FUNCTION_BLOCK FB_Cinta_fms203_SFC
VAR_INPUT
    (* SFC-Flags *)
    SFCPause: BOOL;
    SFCReset: BOOL;

    (* Indicadores de sincronizacion *)
    Ack: BOOL := TRUE;
    Execute: BOOL;
    Restore: BOOL;
    Resume: BOOL;
END_VAR
VAR_OUTPUT
    (* Indicadores de sincronizacion *)
    Done: BOOL;
    Ready: BOOL;
    Restored: BOOL := TRUE;
END_VAR
VAR_INPUT
    (* Funcionalidades *)
    Situar: BOOL;
    Transferir: BOOL;

    (* Parametros *)
    TE: TIME := T#1s; (* Tiempo de entrada del pale *)
    TR: TIME := T#1s; (* Tiempo del retenedor *)
    TS: TIME := T#1s; (* Tiempo del separador *)
    TT: TIME := T#1s; (* Tiempo de transferencia del pale *)
    TX: TIME := T#1s; (* Tiempo de salida del pale *)

    (* Entradas *)
    pp: BOOL; (* Presencia de pale *)
    r0: BOOL; (* Retenedor arriba *)
    r1: BOOL; (* Retenedor abajo *)
    s0: BOOL; (* Separador abajo *)
    _s1: BOOL; (* Separador arriba *)
END_VAR
VAR_OUTPUT
    (* Parametros *)
    Situado: BOOL;
    Transferido: BOOL;

    (* Salidas *)
    RUN: BOOL; (* Motor de la cinta activa [KA1] *)
    REV: BOOL; (* Motor de la cinta invierte [KA2] *)
    R_1: BOOL; (* Retenedor de pale baja [R+] *)
    S_1: BOOL; (* Separador de pale sube [S+] *)
END_VAR
VAR
END_VAR

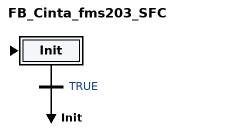
INITIAL_STEP Init:
END_STEP
TRANSITION FROM Init TO Init
    := TRUE;
END_TRANSITION

END_FUNCTION_BLOCK

(* stored: Version 1.1.0.1, ProductVersion 3.1.4024.11
   POU FB_Cinta_fms203_SFC: Id {88efb304-102a-4cc2-bf81-f506df393e08}, SpecialFunc None *)
